// TIA Portal project "Konvenyör Bandı Çalışması SCADA PLCSIM FABRICA.IO Baglantısı_V15.1" (V15.1)
// Vorlageprojekt für das Buch mit Zielsystem S7-1200

(* hardware
DEVICE "S7-1200-Station_1"  S7-1200 Station
   slot 0: "Baugruppenträger_0"  Rack  V1.0
   slot 1: "PLC_1"  CPU 1211C DC/DC/DC  6ES7 211-1AE40-0XB0  V4.1
DEVICE "PC-System_1"  SIMATIC PC station
   slot 0: "SIMATIC PC station"  Rail  SIMATIC PC-Station  V1.0
      slot 125: "Stationmanager"  Station_Manager  V6.0.4
   slot 1: "HMI_RT_1"  WinCC RT Advanced  6AV2 104-0xxxx-xxxx  15.1.0.0
      slot 33792: "Host interface"  Host interface
   slot 2: "IE general_1"  IE General  IE_CP  V8.2.0
*)

// ===== PLC "PLC_1"  CPU 1211C DC/DC/DC =====

VAR_GLOBAL   // PLC tag table "plc_tags"
   "start_buttonu" AT %M5.1 : Bool;
   "stop_butonu" AT %M5.0 : Bool;
   "sistem_devrede" AT %M5.2 : Bool;
   "sistem_calis" AT %Q0.0 : Bool;
   "jog_butonu" AT %M5.4 : Bool;
END_VAR

FUNCTION "MHJ-PLC-Lab-Function-S71200" : Void   // FC9000, SCL
{ S7_Optimized_Access := 'TRUE' }
VERSION : 0.1
   VAR_TEMP
      rdTimeReturn : Int;
      outputTime : DTL;
      SyncVal : Byte;
      forVal : Int;
      forVal_2 : Int;
      Value : Byte;
   END_VAR
   VAR CONSTANT
      CompVal : Byte := 16#34;
      Value_01 : Byte := 16#11;
      Value_01_DW : DWord := 16#A165_D992;
      Value_02_DW : DWord := 16#58BE_4401;
   END_VAR
BEGIN

   #Value:=PEEK(area := 16#82,
        dbNumber := 0,
        byteOffset := 511);
   #Value := #Value + 1;

   POKE(area := 16#82,
        dbNumber := 0,
        byteOffset := 511,
        value := #Value);

   POKE(area:=16#81,
        dbNumber:=0,
        byteOffset:=1016,
        value:=#Value_01_DW);
   POKE(area := 16#81,
        dbNumber := 0,
        byteOffset := 1020,
        value := #Value_02_DW);

   POKE(area := 16#81,
        dbNumber := 0,
        byteOffset := 511,
        value := B#16#00);

   FOR #forVal := 0 TO 120 DO
       FOR #forVal_2:=0 TO 10 DO
           #rdTimeReturn:=RD_SYS_T(#outputTime);
           #rdTimeReturn := WR_SYS_T(#outputTime);
           #rdTimeReturn := RD_SYS_T(#outputTime);
           #rdTimeReturn := WR_SYS_T(#outputTime);
       END_FOR;
       #SyncVal:= PEEK(area := 16#81,
                      dbNumber := 0,
                      byteOffset := 511);
       IF #SyncVal = #CompVal THEN
          GOTO M_1;
       END_IF;
   END_FOR;
   RETURN;

   M_1:
   POKE(area := 16#81,
        dbNumber := 0,
        byteOffset := 511,
        value := B#16#0);
END_FUNCTION

ORGANIZATION_BLOCK "Main"   // OB1, LAD, ProgramCycle
TITLE = "Main Program Sweep (Cycle)"
{ S7_Optimized_Access := 'TRUE' }
VERSION : 0.1
   VAR_INPUT
      Initial_Call : Bool;   // Initial call of this OB
      Remanence : Bool;   // =True, if remanent data are available
   END_VAR
BEGIN

REGION Network 1: Konnektierungsbaustein für PLC-Lab
   // Im Netzwerk 1 wird der Konnektierungsbaustein für PLC-Lab aufgerufen.
   // Dieser Aufruf darf nicht entfernt werden!
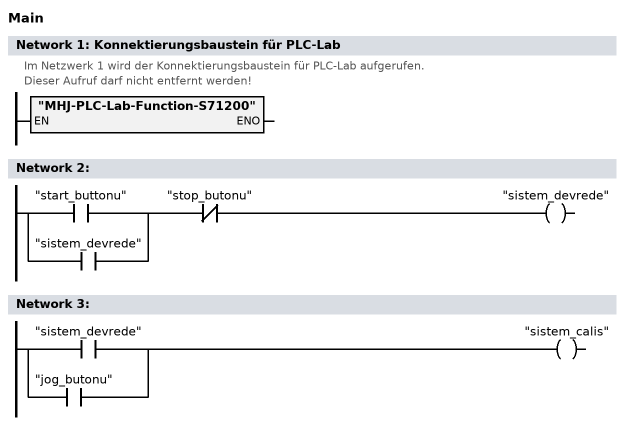
   RUNG wire#powerrail
      "MHJ-PLC-Lab-Function-S71200"()
   END_RUNG
   // the same network as SCL:
   "MHJ-PLC-Lab-Function-S71200"();
END_REGION

REGION Network 2
   RUNG wire#powerrail
      Contact( "start_buttonu" )
      wire#w1
      I_Contact( "stop_butonu" )
      Coil( "sistem_devrede" )
   END_RUNG
   RUNG wire#powerrail
      Contact( "sistem_devrede" )
   END_RUNG wire#w1
   // the same network as SCL:
   "sistem_devrede" := ("start_buttonu" OR "sistem_devrede") AND NOT "stop_butonu";
END_REGION

REGION Network 3
   RUNG wire#powerrail
      Contact( "sistem_devrede" )
      wire#w1
      Coil( "sistem_calis" )
   END_RUNG
   RUNG wire#powerrail
      Contact( "jog_butonu" )
   END_RUNG wire#w1
   // the same network as SCL:
   "sistem_calis" := "sistem_devrede" OR "jog_butonu";
END_REGION
END_ORGANIZATION_BLOCK

(* ===== HMI "HMI_RT_1" =====
system functions are stored by id; their names below are inferred from use
connection "HMI_Connection_1": ETHERNET, S7_1200_OMS

HMI tags "scada_tags"
   "HMI_start" : Bool = PLC start_buttonu AT %M5.1, 100 ms
   "HMI_stop" : Bool = PLC stop_butonu AT %M5.0, 100 ms
   "HMI_jog" : Bool = PLC jog_butonu AT %M5.4, 100 ms

screen "konvenyör kontrol" 1024x766
   Button "Button_2" at 430,114 size 177x152; TextOff 'STOP'
      on Release: ResetBit("HMI_stop")
      on Press: SetBit("HMI_stop")
      Appearance <- "HMI_stop"
   Button "Button_1" at 207,113 size 177x152; TextOff 'START'
      on Press: SetBit("HMI_start")
      on Release: ResetBit("HMI_start")
      Appearance <- "HMI_start"
   Button "Button_3" at 654,115 size 177x152; TextOff 'JOG'
      on Release: ResetBit("HMI_jog")
      on Press: SetBit("HMI_jog")
      Appearance <- "HMI_jog"
   TextField "Text field_1" at 324,18 size 356x33; Text 'KONVENYÖR BANT SİSTEMİ'
*)